(* IEC 61131-3 sources: hayabusa-infrastructure-templates/Ansible/scada/openplc/programs, 2 files *)

(* ---- conveyor_interlock.st ---- *)
PROGRAM ConveyorInterlock
VAR
    estop_ok : BOOL;
    photoeye : BOOL;
    motor_run : BOOL;
    fault : BOOL;
END_VAR

fault := NOT estop_ok;
motor_run := estop_ok AND photoeye AND NOT fault;
END_PROGRAM

(* ---- tank_level.st ---- *)
PROGRAM TankLevel
VAR
    level_high : BOOL;
    level_low : BOOL;
    inlet_valve : BOOL;
    outlet_pump : BOOL;
    alarm : BOOL;
END_VAR

(* Simple tank interlock — additive lab example; does not replace example.st *)
inlet_valve := NOT level_high;
outlet_pump := level_high OR (NOT level_low);
alarm := level_high AND level_low;
END_PROGRAM
